TYPE UR_Safety_Bits_Data :
UNION
	idwURRawInputData : DWORD;
	data : stUR_EIO_Safety_Bits_Mapping;
END_UNION
END_TYPE

(* stored: Version 1.1.0.1, ProductVersion 3.1.4024.16
   DUT UR_Safety_Bits_Data: Id {7bd84855-2597-4dcb-bd8f-b311b4b091b2} *)
